FUNCTION_BLOCK ApplierList 
EXTENDS AbstractDisposableContainer 
IMPLEMENTS CNM_CollectionInterfaces.IApplierList
VAR
	myList 				:ArrayList;
END_VAR

METHOD addApplier : CNM_ReturnTypes.SingleExecutionResult
VAR_INPUT
	applier :CNM_CollectionInterfaces.IApplier;
END_VAR
addApplier := THIS^.myList.append(applier);
END_METHOD

METHOD addAppliers : CNM_ReturnTypes.SingleExecutionResult
VAR_INPUT
	appliers :CNM_CollectionInterfaces.ICollection;
END_VAR
addAppliers := THIS^.myList.appendCollection(appliers);
END_METHOD

PROPERTY className : CNM_AbstractObject.ClassName
GET
className := 'ApplierList';
END_GET
END_PROPERTY

METHOD clear : BOOL
VAR_INPUT
END_VAR
THIS^.myList.clear();
END_METHOD

(*

## Short summary

This method is called in the destruct method and is intended to zero all references and interfaces that should not be destructed. 
To delete the collection with all its contents, use deepDestruct() instead of destruct().

.. <legal notes>

legal notes
=================
| SPDX-FileCopyrightText: © 2025 ekvip automation GmbH <info@ekvip.de>
| SPDX-License-Identifier: Apache-2.0
| For details check: Apache-2.0_

.. _Apache-2.0: https://www.apache.org/licenses/LICENSE-2.0

.. </legal notes>

*)
METHOD PROTECTED clearContents
THIS^.myList.clear();
END_METHOD

(*

## Short summary

This property returns the amount of appliers in the list

.. <legal notes>

legal notes
=================
| SPDX-FileCopyrightText: © 2024 ekvip automation GmbH <info@ekvip.de>
| SPDX-License-Identifier: Apache-2.0
| For details check: Apache-2.0_

.. _Apache-2.0: https://www.apache.org/licenses/LICENSE-2.0

.. </legal notes>

*)

PROPERTY count :UDINT
GET
count := THIS^.myList.size;
END_GET
END_PROPERTY

(*

## Short summary

Mark the object as deleted, as it staiys in the memory.

.. <legal notes>

legal notes
=================
| SPDX-FileCopyrightText: © 2022 ekvip automation GmbH <info@ekvip.de>
| SPDX-License-Identifier: Apache-2.0
| For details check: Apache-2.0_

.. _Apache-2.0: https://www.apache.org/licenses/LICENSE-2.0

.. </legal notes>

*)
METHOD FB_Exit : BOOL
VAR_INPUT
	(* TRUE: the exit method is called in order to leave the instance which will be copied afterwards (online change).*)
	bInCopyCode	: BOOL;
END_VAR
IF THIS^.isObjectValid(THIS^.myList) THEN
	THIS^.myList.deepDestruct();
END_IF
END_METHOD

(*

## Short summary

A method to get an applier at the given index.

.. <legal notes>

legal notes
=================
| SPDX-FileCopyrightText: © 2022 ekvip automation GmbH <info@ekvip.de>
| SPDX-License-Identifier: Apache-2.0
| For details check: Apache-2.0_

.. _Apache-2.0: https://www.apache.org/licenses/LICENSE-2.0

.. </legal notes>


**Return:** CNM_ReturnTypes.ExecutionState

*)

METHOD getApplier : CNM_CollectionInterfaces.IApplier
VAR_INPUT
	index	:UDINT;
END_VAR
VAR
	obj :CNM_AbstractObject.IObject;
END_VAR
THIS^.myList.getObjectAt(index := index, object => obj);
__TRY
	__QUERYINTERFACE(obj, getApplier);
__CATCH
	;
__ENDTRY
END_METHOD

PROPERTY list : CNM_CollectionInterfaces.IArrayList
GET
list := this^.myList;
END_GET
END_PROPERTY

END_FUNCTION_BLOCK

(* stored: Version 1.1.0.1, ProductVersion 3.1.4026.12
   POU ApplierList: Id {0da2f14f-881c-4de6-8aa0-5e5d312c6756}, SpecialFunc None
   Method addApplier: Id {68af4618-579b-4b6e-8305-ce0fa06d6b84}
   Method addAppliers: Id {da227758-b8a3-490f-aff3-a889fe750a71}
   Property className: Id {cab85bff-09ff-4f18-8418-6c14d67169a3}
   Get Get: Id {8287f56e-3db3-4ca4-a6a6-7683ef91b264}
   Method clear: Id {ca95ceaf-935c-4b00-8eec-a63d633f06d7}
   Method clearContents: Id {cddb2888-8427-4349-807a-3d9462896379}
   Property count: Id {c3668de9-1fa1-4d0a-bb73-26c8797e8b54}
   Get Get: Id {0c4492a6-c317-47ac-94f7-9def00163ca8}
   Method FB_Exit: Id {ee80e58c-9512-4e2c-aa22-b13f92561591}
   Method getApplier: Id {41c7edc8-21fe-42e7-9c86-c86c7e1c2247}
   Property list: Id {a5ab7c37-2d37-4334-b1cc-e4d77bcd1e69}
   Get Get: Id {7c7a9d45-ea51-4804-b997-fa8fa5ffea14} *)
